(* IEC 61131-3 sources: AXOpen/src/showcase/app/src/IO, 9 files *)

(* ---- HwIdentifierList.st ---- *)
NAMESPACE AXOpen.Showcase
    TYPE HwIdentifierList : ARRAY[0..442] OF UINT :=
            [
                UINT#32,
                UINT#48,
                UINT#51,
                UINT#54,
                UINT#64,
                UINT#65,
                UINT#66,
                UINT#72,
                UINT#73,
                UINT#74,
                UINT#117,
                UINT#120,
                UINT#121,
                UINT#135,
                UINT#256,
                UINT#257,
                UINT#258,
                UINT#259,
                UINT#260,
                UINT#261,
                UINT#262,
                UINT#263,
                UINT#264,
                UINT#265,
                UINT#266,
                UINT#267,
                UINT#268,
                UINT#269,
                UINT#270,
                UINT#271,
                UINT#272,
                UINT#273,
                UINT#274,
                UINT#275,
                UINT#276,
                UINT#277,
                UINT#278,
                UINT#279,
                UINT#280,
                UINT#281,
                UINT#282,
                UINT#283,
                UINT#284,
                UINT#285,
                UINT#286,
                UINT#287,
                UINT#288,
                UINT#289,
                UINT#290,
                UINT#291,
                UINT#292,
                UINT#293,
                UINT#294,
                UINT#295,
                UINT#296,
                UINT#297,
                UINT#298,
                UINT#299,
                UINT#300,
                UINT#301,
                UINT#302,
                UINT#303,
                UINT#304,
                UINT#305,
                UINT#306,
                UINT#307,
                UINT#308,
                UINT#309,
                UINT#310,
                UINT#311,
                UINT#312,
                UINT#313,
                UINT#314,
                UINT#315,
                UINT#316,
                UINT#317,
                UINT#318,
                UINT#319,
                UINT#320,
                UINT#321,
                UINT#322,
                UINT#323,
                UINT#324,
                UINT#325,
                UINT#326,
                UINT#327,
                UINT#328,
                UINT#329,
                UINT#330,
                UINT#331,
                UINT#332,
                UINT#333,
                UINT#334,
                UINT#335,
                UINT#336,
                UINT#337,
                UINT#338,
                UINT#339,
                UINT#340,
                UINT#341,
                UINT#342,
                UINT#343,
                UINT#344,
                UINT#345,
                UINT#346,
                UINT#347,
                UINT#348,
                UINT#349,
                UINT#350,
                UINT#351,
                UINT#352,
                UINT#353,
                UINT#354,
                UINT#355,
                UINT#356,
                UINT#357,
                UINT#358,
                UINT#359,
                UINT#360,
                UINT#361,
                UINT#362,
                UINT#363,
                UINT#364,
                UINT#365,
                UINT#366,
                UINT#367,
                UINT#368,
                UINT#369,
                UINT#370,
                UINT#371,
                UINT#372,
                UINT#373,
                UINT#374,
                UINT#375,
                UINT#376,
                UINT#377,
                UINT#378,
                UINT#379,
                UINT#380,
                UINT#381,
                UINT#382,
                UINT#383,
                UINT#384,
                UINT#385,
                UINT#386,
                UINT#387,
                UINT#388,
                UINT#389,
                UINT#390,
                UINT#391,
                UINT#392,
                UINT#393,
                UINT#394,
                UINT#395,
                UINT#396,
                UINT#397,
                UINT#398,
                UINT#399,
                UINT#400,
                UINT#401,
                UINT#402,
                UINT#403,
                UINT#404,
                UINT#405,
                UINT#406,
                UINT#407,
                UINT#408,
                UINT#409,
                UINT#410,
                UINT#411,
                UINT#412,
                UINT#413,
                UINT#414,
                UINT#415,
                UINT#416,
                UINT#417,
                UINT#418,
                UINT#419,
                UINT#420,
                UINT#421,
                UINT#422,
                UINT#423,
                UINT#424,
                UINT#425,
                UINT#426,
                UINT#427,
                UINT#428,
                UINT#429,
                UINT#430,
                UINT#431,
                UINT#432,
                UINT#433,
                UINT#434,
                UINT#435,
                UINT#436,
                UINT#437,
                UINT#438,
                UINT#439,
                UINT#440,
                UINT#441,
                UINT#442,
                UINT#443,
                UINT#444,
                UINT#445,
                UINT#446,
                UINT#447,
                UINT#448,
                UINT#449,
                UINT#450,
                UINT#451,
                UINT#452,
                UINT#453,
                UINT#454,
                UINT#455,
                UINT#456,
                UINT#457,
                UINT#458,
                UINT#459,
                UINT#460,
                UINT#461,
                UINT#462,
                UINT#463,
                UINT#464,
                UINT#465,
                UINT#466,
                UINT#467,
                UINT#468,
                UINT#469,
                UINT#470,
                UINT#471,
                UINT#472,
                UINT#473,
                UINT#474,
                UINT#475,
                UINT#476,
                UINT#477,
                UINT#478,
                UINT#479,
                UINT#480,
                UINT#481,
                UINT#482,
                UINT#483,
                UINT#484,
                UINT#485,
                UINT#486,
                UINT#487,
                UINT#488,
                UINT#489,
                UINT#490,
                UINT#491,
                UINT#492,
                UINT#493,
                UINT#494,
                UINT#495,
                UINT#496,
                UINT#497,
                UINT#498,
                UINT#499,
                UINT#500,
                UINT#501,
                UINT#502,
                UINT#503,
                UINT#504,
                UINT#505,
                UINT#506,
                UINT#507,
                UINT#508,
                UINT#509,
                UINT#510,
                UINT#511,
                UINT#512,
                UINT#513,
                UINT#514,
                UINT#515,
                UINT#516,
                UINT#517,
                UINT#518,
                UINT#519,
                UINT#520,
                UINT#521,
                UINT#522,
                UINT#523,
                UINT#524,
                UINT#525,
                UINT#526,
                UINT#527,
                UINT#528,
                UINT#529,
                UINT#530,
                UINT#531,
                UINT#532,
                UINT#533,
                UINT#534,
                UINT#535,
                UINT#536,
                UINT#537,
                UINT#538,
                UINT#539,
                UINT#540,
                UINT#541,
                UINT#542,
                UINT#543,
                UINT#544,
                UINT#545,
                UINT#546,
                UINT#547,
                UINT#548,
                UINT#549,
                UINT#550,
                UINT#551,
                UINT#552,
                UINT#553,
                UINT#554,
                UINT#555,
                UINT#556,
                UINT#557,
                UINT#558,
                UINT#559,
                UINT#560,
                UINT#561,
                UINT#562,
                UINT#563,
                UINT#564,
                UINT#565,
                UINT#566,
                UINT#567,
                UINT#568,
                UINT#569,
                UINT#570,
                UINT#571,
                UINT#572,
                UINT#573,
                UINT#574,
                UINT#575,
                UINT#576,
                UINT#577,
                UINT#578,
                UINT#579,
                UINT#580,
                UINT#581,
                UINT#582,
                UINT#583,
                UINT#584,
                UINT#585,
                UINT#586,
                UINT#587,
                UINT#588,
                UINT#589,
                UINT#590,
                UINT#591,
                UINT#592,
                UINT#593,
                UINT#594,
                UINT#595,
                UINT#596,
                UINT#597,
                UINT#598,
                UINT#599,
                UINT#600,
                UINT#601,
                UINT#602,
                UINT#603,
                UINT#604,
                UINT#605,
                UINT#606,
                UINT#607,
                UINT#608,
                UINT#609,
                UINT#610,
                UINT#611,
                UINT#612,
                UINT#613,
                UINT#614,
                UINT#615,
                UINT#616,
                UINT#617,
                UINT#618,
                UINT#619,
                UINT#620,
                UINT#621,
                UINT#622,
                UINT#623,
                UINT#624,
                UINT#625,
                UINT#626,
                UINT#627,
                UINT#628,
                UINT#629,
                UINT#630,
                UINT#631,
                UINT#632,
                UINT#633,
                UINT#634,
                UINT#635,
                UINT#636,
                UINT#637,
                UINT#638,
                UINT#639,
                UINT#640,
                UINT#641,
                UINT#642,
                UINT#643,
                UINT#644,
                UINT#645,
                UINT#646,
                UINT#647,
                UINT#648,
                UINT#649,
                UINT#650,
                UINT#651,
                UINT#652,
                UINT#653,
                UINT#654,
                UINT#655,
                UINT#656,
                UINT#657,
                UINT#658,
                UINT#659,
                UINT#660,
                UINT#661,
                UINT#662,
                UINT#663,
                UINT#664,
                UINT#665,
                UINT#666,
                UINT#667,
                UINT#668,
                UINT#669,
                UINT#670,
                UINT#671,
                UINT#672,
                UINT#673,
                UINT#674,
                UINT#675,
                UINT#676,
                UINT#677,
                UINT#678,
                UINT#679,
                UINT#680,
                UINT#681,
                UINT#682,
                UINT#683,
                UINT#684
    ];
END_TYPE
END_NAMESPACE

(* ---- HwIdentifiers.st ---- *)
NAMESPACE AXOpen.Showcase
    TYPE
        HwIdentifiers : UINT
        (
            plc_line_HwID := UINT#32,
            plc_line_plc_line_HwID := UINT#48,
            plc_line_plc_line_Card_reader_writer_1_HwID := UINT#51,
            plc_line_plc_line_CPU_display_1_HwID := UINT#54,
            plc_line_plc_line_PROFINET_interface_1_HwID := UINT#64,
            plc_line_plc_line_PROFINET_interface_1_Port_1_HwID := UINT#65,
            plc_line_plc_line_PROFINET_interface_1_Port_2_HwID := UINT#66,
            plc_line_plc_line_PROFINET_interface_2_HwID := UINT#72,
            plc_line_plc_line_PROFINET_interface_2_Port_3_HwID := UINT#73,
            plc_line_plc_line_PROFINET_interface_2_Port_4_HwID := UINT#74,
            plc_line_plc_line_OPC_UA_1_HwID := UINT#117,
            plc_line_plc_line_PROFINET_interface_GBIT_3_HwID := UINT#120,
            plc_line_plc_line_PROFINET_interface_GBIT_3_Port_5_HwID := UINT#121,
            plc_line_plc_line_Virtual_communication_interface_HwID := UINT#135,
            profinet_plc_line_HwID := UINT#256,
            smc_ex260_spn_32_smc_ex260_spn_32_Interface_HwID := UINT#257,
            smc_ex260_spn_32_HwID := UINT#258,
            smc_ex260_spn_32_smc_ex260_spn_32_Interface_Port_1_HwID := UINT#259,
            smc_ex260_spn_32_smc_ex260_spn_32_Interface_Port_2_HwID := UINT#260,
            smc_ex260_spn_32_Rack_HwID := UINT#261,
            smc_ex260_spn_32_smc_ex260_spn_32_HwID := UINT#262,
            smc_ex260_spn_32_smc_ex260_spn_32_Outputs32_4_byte__Output_HwID := UINT#263,
            smc_ex260_spn_32_smc_ex260_spn_32_EX260_SPN_1_2_HwID := UINT#264,
            smc_ex260_spn_16_smc_ex260_spn_16_Interface_HwID := UINT#265,
            smc_ex260_spn_16_HwID := UINT#266,
            smc_ex260_spn_16_smc_ex260_spn_16_Interface_Port_1_HwID := UINT#267,
            smc_ex260_spn_16_smc_ex260_spn_16_Interface_Port_2_HwID := UINT#268,
            smc_ex260_spn_16_Rack_HwID := UINT#269,
            smc_ex260_spn_16_smc_ex260_spn_16_HwID := UINT#270,
            smc_ex260_spn_16_smc_ex260_spn_16_Outputs16_2_byte__Output_HwID := UINT#271,
            smc_ex260_spn_16_smc_ex260_spn_16_EX260_SPN_3_4_HwID := UINT#272,
            aes_pnio_aes_pnio_PN_IO_HwID := UINT#273,
            aes_pnio_HwID := UINT#274,
            aes_pnio_aes_pnio_PN_IO_Port_1_HwID := UINT#275,
            aes_pnio_aes_pnio_PN_IO_Port_2_HwID := UINT#276,
            aes_pnio_Rack_HwID := UINT#277,
            aes_pnio_aes_pnio_HwID := UINT#278,
            aes_pnio_Slot_1_Valve_driver_4_valves_4_HwID := UINT#279,
            aes_pnio_aes_pnio_AES_Modul_HwID := UINT#280,
            rf186c_cyc_rf186c_cyc_profinet_HwID := UINT#281,
            rf186c_cyc_HwID := UINT#282,
            rf186c_cyc_rf186c_cyc_profinet_Port_1_HwID := UINT#283,
            rf186c_cyc_rf186c_cyc_profinet_Port_2_HwID := UINT#284,
            rf186c_cyc_Rack_HwID := UINT#285,
            rf186c_cyc_rf186c_cyc_HwID := UINT#286,
            rf186c_cyc_RF340R_1_Reader_128_byte__cyclic_io_communication_HwID := UINT#287,
            rf186c_cyc_RF260R_1_Reader_32_byte__cyclic_io_communication_HwID := UINT#288,
            rf186c_cyc_rf186c_cyc_CM_Communication_HwID := UINT#289,
            rf186c_cyc_rf186c_cyc_RF186C_cyc_V2_2_HwID := UINT#290,
            et200sp_CM_4xIO_Link_RF200_et200sp_CM_4xIO_Link_RF200_profinet_HwID := UINT#291,
            et200sp_CM_4xIO_Link_RF200_HwID := UINT#292,
            et200sp_CM_4xIO_Link_RF200_et200sp_CM_4xIO_Link_RF200_Port_1_HwID := UINT#293,
            et200sp_CM_4xIO_Link_RF200_et200sp_CM_4xIO_Link_RF200_Port_2_HwID := UINT#294,
            et200sp_CM_4xIO_Link_RF200_Rack_HwID := UINT#295,
            et200sp_CM_4xIO_Link_RF200_et200sp_CM_4xIO_Link_RF200_HwID := UINT#296,
            et200sp_CM_4xIO_Link_RF200_Server_module_V1_1_Server_module_V1_1_0_bytes_HwID := UINT#297,
            et200sp_CM_4xIO_Link_RF200_CM_4xIO_Link_V2_2_144I_128O_1_CM_4xIO_Link_V2_2_144I_128O_HwID := UINT#298,
            et200sp_CM_4xIO_Link_RF200_et200sp_CM_4xIO_Link_RF200_IM_155_6_PN_ST_V4_2_HwID := UINT#299,
            rf186c_rf186c_profinet_HwID := UINT#300,
            rf186c_HwID := UINT#301,
            rf186c_rf186c_profinet_Port_1_HwID := UINT#302,
            rf186c_rf186c_profinet_Port_2_HwID := UINT#303,
            rf186c_Rack_HwID := UINT#304,
            rf186c_rf186c_HwID := UINT#305,
            rf186c_Reader_1__Reader__HwID := UINT#306,
            rf186c_rf186c_CM_1__Communication__HwID := UINT#307,
            rf186c_rf186c_RF186C_V2_x_HwID := UINT#308,
            et200sp_et200sp_profinet_HwID := UINT#309,
            et200sp_HwID := UINT#310,
            et200sp_et200sp_Port_1_HwID := UINT#311,
            et200sp_et200sp_Port_2_HwID := UINT#312,
            et200sp_Rack_HwID := UINT#313,
            et200sp_et200sp_HwID := UINT#314,
            et200sp_Server_module_V1_1_Server_module_V1_1_0_bytes_HwID := UINT#315,
            et200sp_CpPtp_CM_PtP_V2_0_HwID := UINT#316,
            et200sp_et200sp_IM_155_6_PN_ST_V4_2_HwID := UINT#317,
            BNIPNT507005Z040_BNIPNT507005Z040_profinet_HwID := UINT#318,
            BNIPNT507005Z040_HwID := UINT#319,
            BNIPNT507005Z040_BNIPNT507005Z040_profinet_port_1_M12_HwID := UINT#320,
            BNIPNT507005Z040_BNIPNT507005Z040_profinet_port_2_M12_HwID := UINT#321,
            BNIPNT507005Z040_Rack_HwID := UINT#322,
            BNIPNT507005Z040_BNIPNT507005Z040_HwID := UINT#323,
            BNIPNT507005Z040_BIS_M_4XX_045_1_BIS_M_4XX_045_HwID := UINT#324,
            BNIPNT507005Z040_Standard_I_O_4_Standard_I_O_HwID := UINT#325,
            BNIPNT507005Z040_Standard_I_O_3_Standard_I_O_HwID := UINT#326,
            BNIPNT507005Z040_Standard_I_O_2_Standard_I_O_HwID := UINT#327,
            BNIPNT507005Z040_BNIPNT507005Z040_BNI_PNT_507_005_Z040_HwID := UINT#328,
            rexroth_cs351_rexroth_cs351_Interface_HwID := UINT#329,
            rexroth_cs351_HwID := UINT#330,
            rexroth_cs351_rexroth_cs351_Interface_Port_1_HwID := UINT#331,
            rexroth_cs351_Rack_HwID := UINT#332,
            rexroth_cs351_rexroth_cs351_HwID := UINT#333,
            rexroth_cs351_Input_2_word_1_Input_2_word_HwID := UINT#334,
            rexroth_cs351_Input_4_word_16_Input_4_word_HwID := UINT#335,
            rexroth_cs351_Input_4_word_15_Input_4_word_HwID := UINT#336,
            rexroth_cs351_Input_4_word_14_Input_4_word_HwID := UINT#337,
            rexroth_cs351_Input_4_word_13_Input_4_word_HwID := UINT#338,
            rexroth_cs351_Input_4_word_12_Input_4_word_HwID := UINT#339,
            rexroth_cs351_Input_4_word_11_Input_4_word_HwID := UINT#340,
            rexroth_cs351_Input_4_word_10_Input_4_word_HwID := UINT#341,
            rexroth_cs351_Input_4_word_9_Input_4_word_HwID := UINT#342,
            rexroth_cs351_Input_4_word_8_Input_4_word_HwID := UINT#343,
            rexroth_cs351_Input_4_word_7_Input_4_word_HwID := UINT#344,
            rexroth_cs351_Input_4_word_6_Input_4_word_HwID := UINT#345,
            rexroth_cs351_Input_4_word_5_Input_4_word_HwID := UINT#346,
            rexroth_cs351_Input_4_word_4_Input_4_word_HwID := UINT#347,
            rexroth_cs351_Input_4_word_3_Input_4_word_HwID := UINT#348,
            rexroth_cs351_Input_4_word_2_Input_4_word_HwID := UINT#349,
            rexroth_cs351_Input_4_word_1_Input_4_word_HwID := UINT#350,
            rexroth_cs351_Output_2_word_1_Output_2_word_HwID := UINT#351,
            rexroth_cs351_Output_4_word_8_Output_4_word_HwID := UINT#352,
            rexroth_cs351_Output_4_word_7_Output_4_word_HwID := UINT#353,
            rexroth_cs351_Output_4_word_6_Output_4_word_HwID := UINT#354,
            rexroth_cs351_Output_4_word_5_Output_4_word_HwID := UINT#355,
            rexroth_cs351_Output_4_word_4_Output_4_word_HwID := UINT#356,
            rexroth_cs351_Output_4_word_3_Output_4_word_HwID := UINT#357,
            rexroth_cs351_Output_4_word_2_Output_4_word_HwID := UINT#358,
            rexroth_cs351_Output_4_word_1_Output_4_word_HwID := UINT#359,
            rexroth_cs351_rexroth_cs351_DAP_V2_0_HwID := UINT#360,
            rexroth_press_rexroth_press_PN_IO_HwID := UINT#361,
            rexroth_press_HwID := UINT#362,
            rexroth_press_rexroth_press_PN_IO_Port_1_HwID := UINT#363,
            rexroth_press_rexroth_press_PN_IO_Port_2_HwID := UINT#364,
            rexroth_press_Rack_HwID := UINT#365,
            rexroth_press_rexroth_press_HwID := UINT#366,
            rexroth_press_Output_21_Words_ID_OutMod_21Words_HwID := UINT#367,
            rexroth_press_Input_24_Words_ID_InMod_24Words_HwID := UINT#368,
            rexroth_press_ParamCh_5Words_ID_PaCh_5Words_HwID := UINT#369,
            rexroth_press_F_Modul_not_used_ID_FMod_NotUsed_HwID := UINT#370,
            rexroth_press_rexroth_press_DAP_1_HwID := UINT#371,
            dukaneiqauto_dukaneiqauto_Interface_HwID := UINT#372,
            dukaneiqauto_HwID := UINT#373,
            dukaneiqauto_dukaneiqauto_Interface_Port_1_HwID := UINT#374,
            dukaneiqauto_dukaneiqauto_Interface_Port_2_HwID := UINT#375,
            dukaneiqauto_Rack_HwID := UINT#376,
            dukaneiqauto_dukaneiqauto_HwID := UINT#377,
            dukaneiqauto_PLC_to_iQ_Outputs_PLC_to_iQ_Outputs_HwID := UINT#378,
            dukaneiqauto_iQ_to_PLC_Inputs_iQ_to_PLC_Inputs_HwID := UINT#379,
            dukaneiqauto_dukaneiqauto_DAP_HwID := UINT#380,
            desoutter_cvic_ii_desoutter_cvic_ii_Interface_HwID := UINT#381,
            desoutter_cvic_ii_HwID := UINT#382,
            desoutter_cvic_ii_desoutter_cvic_ii_Interface_Port_1_HwID := UINT#383,
            desoutter_cvic_ii_Rack_HwID := UINT#384,
            desoutter_cvic_ii_desoutter_cvic_ii_HwID := UINT#385,
            desoutter_cvic_ii_Output_1_byte_2_Output_1_byte_HwID := UINT#386,
            desoutter_cvic_ii_Output_1_byte_1_Output_1_byte_HwID := UINT#387,
            desoutter_cvic_ii_Input_1_word_2_Input_1_word_HwID := UINT#388,
            desoutter_cvic_ii_Input_2_word_2_Input_2_word_HwID := UINT#389,
            desoutter_cvic_ii_Input_1_word_1_Input_1_word_HwID := UINT#390,
            desoutter_cvic_ii_Input_2_word_1_Input_2_word_HwID := UINT#391,
            desoutter_cvic_ii_Input_1_byte_2_Input_1_byte_HwID := UINT#392,
            desoutter_cvic_ii_Input_1_byte_1_Input_1_byte_HwID := UINT#393,
            desoutter_cvic_ii_desoutter_cvic_ii_RT_HwID := UINT#394,
            zebra_zebra_Interface_HwID := UINT#395,
            zebra_HwID := UINT#396,
            zebra_zebra_Interface_Port_1_HwID := UINT#397,
            zebra_Rack_HwID := UINT#398,
            zebra_zebra_HwID := UINT#399,
            zebra_Data88Bin6Bout_Data_and_Transfer_Control_v2_HwID := UINT#400,
            zebra_zebra_EA3600_PIO_Interface_HwID := UINT#401,
            keyence_iv3_keyence_iv3_Interface_HwID := UINT#402,
            keyence_iv3_HwID := UINT#403,
            keyence_iv3_keyence_iv3_Interface_Port_1_HwID := UINT#404,
            keyence_iv3_Rack_HwID := UINT#405,
            keyence_iv3_keyence_iv3_HwID := UINT#406,
            keyence_iv3_DeviceResultBits_2_Device_Result_Bits_HwID := UINT#407,
            keyence_iv3_ToolResult_64_Tool_Result_HwID := UINT#408,
            keyence_iv3_ToolResult_63_Tool_Result_HwID := UINT#409,
            keyence_iv3_ToolResult_62_Tool_Result_HwID := UINT#410,
            keyence_iv3_ToolResult_61_Tool_Result_HwID := UINT#411,
            keyence_iv3_ToolResult_60_Tool_Result_HwID := UINT#412,
            keyence_iv3_ToolResult_59_Tool_Result_HwID := UINT#413,
            keyence_iv3_ToolResult_58_Tool_Result_HwID := UINT#414,
            keyence_iv3_ToolResult_57_Tool_Result_HwID := UINT#415,
            keyence_iv3_ToolResult_56_Tool_Result_HwID := UINT#416,
            keyence_iv3_ToolResult_55_Tool_Result_HwID := UINT#417,
            keyence_iv3_ToolResult_54_Tool_Result_HwID := UINT#418,
            keyence_iv3_ToolResult_53_Tool_Result_HwID := UINT#419,
            keyence_iv3_ToolResult_52_Tool_Result_HwID := UINT#420,
            keyence_iv3_ToolResult_51_Tool_Result_HwID := UINT#421,
            keyence_iv3_ToolResult_50_Tool_Result_HwID := UINT#422,
            keyence_iv3_ToolResult_49_Tool_Result_HwID := UINT#423,
            keyence_iv3_ToolResult_48_Tool_Result_HwID := UINT#424,
            keyence_iv3_ToolResult_47_Tool_Result_HwID := UINT#425,
            keyence_iv3_ToolResult_46_Tool_Result_HwID := UINT#426,
            keyence_iv3_ToolResult_45_Tool_Result_HwID := UINT#427,
            keyence_iv3_ToolResult_44_Tool_Result_HwID := UINT#428,
            keyence_iv3_ToolResult_43_Tool_Result_HwID := UINT#429,
            keyence_iv3_ToolResult_42_Tool_Result_HwID := UINT#430,
            keyence_iv3_ToolResult_41_Tool_Result_HwID := UINT#431,
            keyence_iv3_ToolResult_40_Tool_Result_HwID := UINT#432,
            keyence_iv3_ToolResult_39_Tool_Result_HwID := UINT#433,
            keyence_iv3_ToolResult_38_Tool_Result_HwID := UINT#434,
            keyence_iv3_ToolResult_37_Tool_Result_HwID := UINT#435,
            keyence_iv3_ToolResult_36_Tool_Result_HwID := UINT#436,
            keyence_iv3_ToolResult_35_Tool_Result_HwID := UINT#437,
            keyence_iv3_ToolResult_34_Tool_Result_HwID := UINT#438,
            keyence_iv3_ToolResult_33_Tool_Result_HwID := UINT#439,
            keyence_iv3_ToolResult_32_Tool_Result_HwID := UINT#440,
            keyence_iv3_ToolResult_31_Tool_Result_HwID := UINT#441,
            keyence_iv3_ToolResult_30_Tool_Result_HwID := UINT#442,
            keyence_iv3_ToolResult_29_Tool_Result_HwID := UINT#443,
            keyence_iv3_ToolResult_28_Tool_Result_HwID := UINT#444,
            keyence_iv3_ToolResult_27_Tool_Result_HwID := UINT#445,
            keyence_iv3_ToolResult_26_Tool_Result_HwID := UINT#446,
            keyence_iv3_ToolResult_25_Tool_Result_HwID := UINT#447,
            keyence_iv3_ToolResult_24_Tool_Result_HwID := UINT#448,
            keyence_iv3_ToolResult_23_Tool_Result_HwID := UINT#449,
            keyence_iv3_ToolResult_22_Tool_Result_HwID := UINT#450,
            keyence_iv3_ToolResult_21_Tool_Result_HwID := UINT#451,
            keyence_iv3_ToolResult_20_Tool_Result_HwID := UINT#452,
            keyence_iv3_ToolResult_19_Tool_Result_HwID := UINT#453,
            keyence_iv3_ToolResult_18_Tool_Result_HwID := UINT#454,
            keyence_iv3_ToolResult_17_Tool_Result_HwID := UINT#455,
            keyence_iv3_ToolResult_16_Tool_Result_HwID := UINT#456,
            keyence_iv3_ToolResult_15_Tool_Result_HwID := UINT#457,
            keyence_iv3_ToolResult_14_Tool_Result_HwID := UINT#458,
            keyence_iv3_ToolResult_13_Tool_Result_HwID := UINT#459,
            keyence_iv3_ToolResult_12_Tool_Result_HwID := UINT#460,
            keyence_iv3_ToolResult_11_Tool_Result_HwID := UINT#461,
            keyence_iv3_ToolResult_10_Tool_Result_HwID := UINT#462,
            keyence_iv3_ToolResult_9_Tool_Result_HwID := UINT#463,
            keyence_iv3_ToolResult_8_Tool_Result_HwID := UINT#464,
            keyence_iv3_ToolResult_7_Tool_Result_HwID := UINT#465,
            keyence_iv3_ToolResult_6_Tool_Result_HwID := UINT#466,
            keyence_iv3_ToolResult_5_Tool_Result_HwID := UINT#467,
            keyence_iv3_ToolResult_4_Tool_Result_HwID := UINT#468,
            keyence_iv3_ToolResult_3_Tool_Result_HwID := UINT#469,
            keyence_iv3_ToolResult_2_Tool_Result_HwID := UINT#470,
            keyence_iv3_ToolResult_1_Tool_Result_HwID := UINT#471,
            keyence_iv3_PositionAdjustResult_Position_Adjust_Result_HwID := UINT#472,
            keyence_iv3_DeviceStatistics_Device_Statistics_HwID := UINT#473,
            keyence_iv3_DeviceStatusWords_Device_Status_Words_HwID := UINT#474,
            keyence_iv3_DeviceResultBits_1_Device_Result_Bits_HwID := UINT#475,
            keyence_iv3_CommandStatusBits_Command_Status_Bits_HwID := UINT#476,
            keyence_iv3_CommandControl_Command_Control_HwID := UINT#477,
            keyence_iv3_keyence_iv3_IV3_XXXX_HwID := UINT#478,
            keyence_sr_1000_keyence_sr_1000_Interface_HwID := UINT#479,
            keyence_sr_1000_HwID := UINT#480,
            keyence_sr_1000_keyence_sr_1000_Interface_Port_1_HwID := UINT#481,
            keyence_sr_1000_Rack_HwID := UINT#482,
            keyence_sr_1000_keyence_sr_1000_HwID := UINT#483,
            keyence_sr_1000_UserData_128_User_Data_128Byte_HwID := UINT#484,
            keyence_sr_1000_ParameterBank_Parameter_Bank_Number_HwID := UINT#485,
            keyence_sr_1000_CompletionClearControl_Completion_Clear_Control_Bits_HwID := UINT#486,
            keyence_sr_1000_OperationInstructionControl_Operation_instruction_Control_Bits_HwID := UINT#487,
            keyence_sr_1000_LatchAndErrorClearControl_Latch_and_Error_Clear_Control_Bits_HwID := UINT#488,
            keyence_sr_1000_ResultData_128_Read_Data_128Byte_HwID := UINT#489,
            keyence_sr_1000_OperationResultStatus_Operation_Result_Status_HwID := UINT#490,
            keyence_sr_1000_MatchingLevelAndTotalEvaluationGradeStatus_Matching_Level_and_Total_Evaluation_Grade_Status_HwID := UINT#491,
            keyence_sr_1000_UnstableReadStatus_Unstable_Read_Status_Bits_HwID := UINT#492,
            keyence_sr_1000_TerminalStatus_Terminal_Status_Bits_HwID := UINT#493,
            keyence_sr_1000_ErrorStatus_Error_Status_Bits_HwID := UINT#494,
            keyence_sr_1000_CompletionStatus_Completion_Status_Bits_HwID := UINT#495,
            keyence_sr_1000_BusyStatus_BUSY_Status_Bits_HwID := UINT#496,
            keyence_sr_1000_HandshakeAndGeneralErrorStatus_Handshake_and_General_Error_Status_Bits_HwID := UINT#497,
            keyence_sr_1000_keyence_sr_1000_SR_1000X_HwID := UINT#498,
            keyence_sr_750_keyence_sr_750_Interface_HwID := UINT#499,
            keyence_sr_750_HwID := UINT#500,
            keyence_sr_750_keyence_sr_750_Interface_Port_1_HwID := UINT#501,
            keyence_sr_750_Rack_HwID := UINT#502,
            keyence_sr_750_keyence_sr_750_HwID := UINT#503,
            keyence_sr_750_UserData_128_User_Data_128Byte_HwID := UINT#504,
            keyence_sr_750_ParameterBank_Parameter_Bank_Number_HwID := UINT#505,
            keyence_sr_750_CompletionClearControl_Completion_Clear_Control_Bits_HwID := UINT#506,
            keyence_sr_750_OperationInstructionControl_Operation_instruction_Control_Bits_HwID := UINT#507,
            keyence_sr_750_LatchAndErrorClearControl_Latch_and_Error_Clear_Control_Bits_HwID := UINT#508,
            keyence_sr_750_ResultData_128_Read_Data_128Byte_HwID := UINT#509,
            keyence_sr_750_OperationResultStatus_Operation_Result_Status_HwID := UINT#510,
            keyence_sr_750_MatchingLevelAndTotalEvaluationGradeStatus_Matching_Level_and_Total_Evaluation_Grade_Status_HwID := UINT#511,
            keyence_sr_750_UnstableReadStatus_Unstable_Read_Status_Bits_HwID := UINT#512,
            keyence_sr_750_TerminalStatus_Terminal_Status_Bits_HwID := UINT#513,
            keyence_sr_750_ErrorStatus_Error_Status_Bits_HwID := UINT#514,
            keyence_sr_750_CompletionStatus_Completion_Status_Bits_HwID := UINT#515,
            keyence_sr_750_BusyStatus_BUSY_Status_Bits_HwID := UINT#516,
            keyence_sr_750_HandshakeAndGeneralErrorStatus_Handshake_and_General_Error_Status_Bits_HwID := UINT#517,
            keyence_sr_750_keyence_sr_750_SR_75X_HwID := UINT#518,
            vision_pro_vision_pro_Interface_HwID := UINT#519,
            vision_pro_HwID := UINT#520,
            vision_pro_vision_pro_Interface_Port_1_HwID := UINT#521,
            vision_pro_Rack_HwID := UINT#522,
            vision_pro_vision_pro_HwID := UINT#523,
            vision_pro_Result_Data_64_bytes_1_Results_64_bytes_HwID := UINT#524,
            vision_pro_Result_Data_240_bytes_5_Results_240_bytes_HwID := UINT#525,
            vision_pro_Result_Data_240_bytes_4_Results_240_bytes_HwID := UINT#526,
            vision_pro_Result_Data_240_bytes_3_Results_240_bytes_HwID := UINT#527,
            vision_pro_Result_Data_240_bytes_2_Results_240_bytes_HwID := UINT#528,
            vision_pro_User_Data_64_bytes_1_User_Data_64_bytes_HwID := UINT#529,
            vision_pro_User_Data_240_bytes_5_User_Data_240_bytes_HwID := UINT#530,
            vision_pro_User_Data_240_bytes_4_User_Data_240_bytes_HwID := UINT#531,
            vision_pro_User_Data_240_bytes_3_User_Data_240_bytes_HwID := UINT#532,
            vision_pro_User_Data_240_bytes_2_User_Data_240_bytes_HwID := UINT#533,
            vision_pro_Result_Data_240_bytes_1_Results_240_bytes_HwID := UINT#534,
            vision_pro_User_Data_240_bytes_1_User_Data_240_bytes_HwID := UINT#535,
            vision_pro_Engine_Control_4_Engine_Control_HwID := UINT#536,
            vision_pro_Engine_Control_3_Engine_Control_HwID := UINT#537,
            vision_pro_Engine_Control_2_Engine_Control_HwID := UINT#538,
            vision_pro_Engine_Control_1_Engine_Control_HwID := UINT#539,
            vision_pro_System_Control_System_Control_HwID := UINT#540,
            vision_pro_vision_pro_Communication_Card_CC24_HwID := UINT#541,
            cognex_insight_2800_cognex_insight_2800_Interface_HwID := UINT#542,
            cognex_insight_2800_HwID := UINT#543,
            cognex_insight_2800_cognex_insight_2800_Interface_Port_1_HwID := UINT#544,
            cognex_insight_2800_Rack_HwID := UINT#545,
            cognex_insight_2800_cognex_insight_2800_HwID := UINT#546,
            cognex_insight_2800_Slot_14_Results_250_bytes_HwID := UINT#547,
            cognex_insight_2800_Slot_13_Results_250_bytes_HwID := UINT#548,
            cognex_insight_2800_Slot_12_Results_250_bytes_HwID := UINT#549,
            cognex_insight_2800_Slot_11_ResultData_250_Results_250_bytes_HwID := UINT#550,
            cognex_insight_2800_Slot_9_User_Data_254_bytes_HwID := UINT#551,
            cognex_insight_2800_Slot_8_User_Data_254_bytes_HwID := UINT#552,
            cognex_insight_2800_Slot_7_User_Data_254_bytes_HwID := UINT#553,
            cognex_insight_2800_Slot_2_Acquisition_Status_HwID := UINT#554,
            cognex_insight_2800_Slot_4_Inspection_Status_HwID := UINT#555,
            cognex_insight_2800_Slot_5_Command_Control_HwID := UINT#556,
            cognex_insight_2800_Slot_6_ExternalEvent_Control_HwID := UINT#557,
            cognex_insight_2800_Slot_3_Inspection_Control_HwID := UINT#558,
            cognex_insight_2800_Slot_1_Acquisition_Control_HwID := UINT#559,
            cognex_insight_2800_cognex_insight_2800_In_Sight_IS28XX_CC_B_HwID := UINT#560,
            cognex_dataman_380_cognex_dataman_380_Interface_HwID := UINT#561,
            cognex_dataman_380_HwID := UINT#562,
            cognex_dataman_380_cognex_dataman_380_Interface_Port_1_HwID := UINT#563,
            cognex_dataman_380_Rack_HwID := UINT#564,
            cognex_dataman_380_cognex_dataman_380_HwID := UINT#565,
            cognex_dataman_380_ResultData_128_Result_Data_128_bytes_HwID := UINT#566,
            cognex_dataman_380_UserData_128_User_Data_128_bytes_HwID := UINT#567,
            cognex_dataman_380_Results_Status_Results_Status_HwID := UINT#568,
            cognex_dataman_380_Acquisition_Status_Acquisition_Status_HwID := UINT#569,
            cognex_dataman_380_Soft_Event_Control_Soft_Event_Control_HwID := UINT#570,
            cognex_dataman_380_Results_Control_Results_Control_HwID := UINT#571,
            cognex_dataman_380_Acquisition_Control_Acquisition_Control_HwID := UINT#572,
            cognex_dataman_380_cognex_dataman_380_DataMan_380_CC_B_HwID := UINT#573,
            cognex_dataman_280_cognex_dataman_280_Interface_HwID := UINT#574,
            cognex_dataman_280_HwID := UINT#575,
            cognex_dataman_280_cognex_dataman_280_Interface_Port_1_HwID := UINT#576,
            cognex_dataman_280_Rack_HwID := UINT#577,
            cognex_dataman_280_cognex_dataman_280_HwID := UINT#578,
            cognex_dataman_280_ResultData_128_Result_Data_128_bytes_HwID := UINT#579,
            cognex_dataman_280_UserData_128_User_Data_128_bytes_HwID := UINT#580,
            cognex_dataman_280_Results_Status_Results_Status_HwID := UINT#581,
            cognex_dataman_280_Acquisition_Status_Acquisition_Status_HwID := UINT#582,
            cognex_dataman_280_Soft_Event_Control_Soft_Event_Control_HwID := UINT#583,
            cognex_dataman_280_Results_Control_Results_Control_HwID := UINT#584,
            cognex_dataman_280_Acquisition_Control_Acquisition_Control_HwID := UINT#585,
            cognex_dataman_280_cognex_dataman_280_DataMan_280_CC_B_HwID := UINT#586,
            cognex_insight_7600_cognex_insight_7600_Interface_HwID := UINT#587,
            cognex_insight_7600_HwID := UINT#588,
            cognex_insight_7600_cognex_insight_7600_Interface_Port_1_HwID := UINT#589,
            cognex_insight_7600_Rack_HwID := UINT#590,
            cognex_insight_7600_cognex_insight_7600_HwID := UINT#591,
            cognex_insight_7600_ResultData_128_Results_128_bytes_HwID := UINT#592,
            cognex_insight_7600_UserData_128_User_Data_128_bytes_HwID := UINT#593,
            cognex_insight_7600_Inspection_Status_Inspection_Status_HwID := UINT#594,
            cognex_insight_7600_Acquisition_Status_Acquisition_Status_HwID := UINT#595,
            cognex_insight_7600_Command_Control_Command_Control_HwID := UINT#596,
            cognex_insight_7600_SoftEvent_Control_SoftEvent_Control_HwID := UINT#597,
            cognex_insight_7600_Inspection_Control_Inspection_Control_HwID := UINT#598,
            cognex_insight_7600_Acquisition_Control_Acquisition_Control_HwID := UINT#599,
            cognex_insight_7600_cognex_insight_7600_In_Sight_IS79XX_IS75XX_CC_B_HwID := UINT#600,
            rexroth_ctrlx_drive_rexroth_ctrlx_drive_XCS_interface_PF30_HwID := UINT#601,
            rexroth_ctrlx_drive_HwID := UINT#602,
            rexroth_ctrlx_drive_rexroth_ctrlx_drive_XCS_interface_PF30_Port_1_HwID := UINT#603,
            rexroth_ctrlx_drive_rexroth_ctrlx_drive_XCS_interface_PF30_Port_2_HwID := UINT#604,
            rexroth_ctrlx_drive_Rack_HwID := UINT#605,
            rexroth_ctrlx_drive_rexroth_ctrlx_drive_HwID := UINT#606,
            rexroth_ctrlx_drive_Outputs_HwID := UINT#607,
            rexroth_ctrlx_drive_Inputs_HwID := UINT#608,
            rexroth_ctrlx_drive_S_0_0386_0_0__Position_controller__Position_actual_value_HwID := UINT#609,
            rexroth_ctrlx_drive_S_0_0535_0_0__Velocity_controller__Velocity_actual_value_HwID := UINT#610,
            rexroth_ctrlx_drive_S_0_0390_0_0__Diagnostic_message__Manufacturer_status_register_HwID := UINT#611,
            rexroth_ctrlx_drive_S_0_0135_0_0__Drive_status_word__Value_HwID := UINT#612,
            rexroth_ctrlx_drive_S_0_0144_0_0__Signal_status_word__Value_HwID := UINT#613,
            rexroth_ctrlx_drive_S_0_1720_0_2__Power_supply_control__Status_word_HwID := UINT#614,
            rexroth_ctrlx_drive_S_0_0084_0_0__Torque_force_feedback_value_HwID := UINT#615,
            rexroth_ctrlx_drive_P_0_0106_0_0__STO_function__Operating_status_HwID := UINT#616,
            rexroth_ctrlx_drive_S_0_0134_0_0__Master_control_word__Value_HwID := UINT#617,
            rexroth_ctrlx_drive_S_0_0260_0_0__Positioning_profile__Acceleration_HwID := UINT#618,
            rexroth_ctrlx_drive_S_0_0282_0_0__Drive_controlled_positioning__Command_value_HwID := UINT#619,
            rexroth_ctrlx_drive_S_0_0359_0_0__Positioning_profile__Deceleration_HwID := UINT#620,
            rexroth_ctrlx_drive_S_0_0259_0_0__Positioning_profile__Profile_velocity_HwID := UINT#621,
            rexroth_ctrlx_drive_S_0_0145_0_0__Signal_control_word__Value_HwID := UINT#622,
            rexroth_ctrlx_drive_S_0_1720_0_1__Power_supply_control__Control_word_HwID := UINT#623,
            rexroth_ctrlx_drive_S_0_0092_0_0__Torque_force_limitation__Limit_value_bipolar_HwID := UINT#624,
            rexroth_ctrlx_drive_S_0_0080_0_0__Torque_force_command_value_HwID := UINT#625,
            rexroth_ctrlx_drive_S_0_0193_0_0__Positioning_jerk_HwID := UINT#626,
            rexroth_ctrlx_drive_rexroth_ctrlx_drive_ctrlX_DRIVE_XCS_HwID := UINT#627,
            rexroth_indradrive_rexroth_indradrive_PN_IO_HwID := UINT#628,
            rexroth_indradrive_HwID := UINT#629,
            rexroth_indradrive_rexroth_indradrive_PN_IO_Port_1_HwID := UINT#630,
            rexroth_indradrive_rexroth_indradrive_PN_IO_Port_2_HwID := UINT#631,
            rexroth_indradrive_Rack_HwID := UINT#632,
            rexroth_indradrive_rexroth_indradrive_HwID := UINT#633,
            rexroth_indradrive_Output_13_Words_ID_OutMod_13Words_HwID := UINT#634,
            rexroth_indradrive_Input_9_Words_ID_InMod_9Words_HwID := UINT#635,
            rexroth_indradrive_ParamCh_5Words_ID_PaCh_5Words_HwID := UINT#636,
            rexroth_indradrive_F_Modul_not_used_ID_FMod_NotUsed_HwID := UINT#637,
            rexroth_indradrive_rexroth_indradrive_DAP_1_HwID := UINT#638,
            festo_cmmtas_festo_cmmtas_PN_IO_Interface_HwID := UINT#639,
            festo_cmmtas_HwID := UINT#640,
            festo_cmmtas_festo_cmmtas_PN_IO_Interface_Port_1_HwID := UINT#641,
            festo_cmmtas_festo_cmmtas_PN_IO_Interface_Port_2_HwID := UINT#642,
            festo_cmmtas_Rack_HwID := UINT#643,
            festo_cmmtas_festo_cmmtas_HwID := UINT#644,
            festo_cmmtas_festo_cmmtas_DoServo_HwID := UINT#645,
            festo_cmmtas_festo_cmmtas_DoServo_Module_Access_Point_HwID := UINT#646,
            festo_cmmtas_festo_cmmtas_empty_submodule_1_HwID := UINT#647,
            festo_cmmtas_empty_submodule_HwID := UINT#648,
            festo_cmmtas_SiemensTelegram111_PZD_12_12_HwID := UINT#649,
            festo_cmmtas_SiemensTelegram750_PZD_4_1_HwID := UINT#650,
            festo_cmmtas_festo_cmmtas_CMMT_AS___MP_HwID := UINT#651,
            ureol2l_ureol2l_Interface_HwID := UINT#652,
            ureol2l_HwID := UINT#653,
            ureol2l_ureol2l_Interface_Port_1_HwID := UINT#654,
            ureol2l_Rack_HwID := UINT#655,
            ureol2l_ureol2l_HwID := UINT#656,
            ureol2l_10_O2T_General_Purpose_Registers_2_10_O2T_General_Purpose_Registers_2_HwID := UINT#657,
            ureol2l_9_O2T_General_Purpose_Registers_1_9_O2T_General_Purpose_Registers_1_HwID := UINT#658,
            ureol2l_8_O2T_Robot_IO_8_O2T_Robot_IO_HwID := UINT#659,
            ureol2l_7_T2O_General_Purpose_Float_Registers_7_T2O_General_Purpose_Float_Registers_HwID := UINT#660,
            ureol2l_6_T2O_General_Purpose_Int_Registers_6_T2O_General_Purpose_Int_Registers_HwID := UINT#661,
            ureol2l_5_T2O_General_Purpose_Bit_Registers_5_T2O_General_Purpose_Bit_Registers_HwID := UINT#662,
            ureol2l_4_T2O_TCP_4_T2O_TCP_HwID := UINT#663,
            ureol2l_3_T2O_Joints_3_T2O_Joints_HwID := UINT#664,
            ureol2l_2_T2O_IO_2_T2O_IO_HwID := UINT#665,
            ureol2l_1_T2O_State_1_T2O_State_HwID := UINT#666,
            ureol2l_ureol2l_V1_0_HwID := UINT#667,
            mitsubishi_tz535_robot_mitsubishi_tz535_robot_Interface_HwID := UINT#668,
            mitsubishi_tz535_robot_HwID := UINT#669,
            mitsubishi_tz535_robot_mitsubishi_tz535_robot_Interface_Port_1_HwID := UINT#670,
            mitsubishi_tz535_robot_mitsubishi_tz535_robot_Interface_Port_2_HwID := UINT#671,
            mitsubishi_tz535_robot_Rack_HwID := UINT#672,
            mitsubishi_tz535_robot_mitsubishi_tz535_robot_HwID := UINT#673,
            mitsubishi_tz535_robot_In_Out_64_byte_In_Out__64_byte_HwID := UINT#674,
            mitsubishi_tz535_robot_mitsubishi_tz535_robot_2D_TZ535_PNPROFINET_IO_HwID := UINT#675,
            kuka_rb2_kuka_rb2_Interface1_HwID := UINT#676,
            kuka_rb2_HwID := UINT#677,
            kuka_rb2_kuka_rb2_Interface1_Port_1_HwID := UINT#678,
            kuka_rb2_kuka_rb2_Interface1_Port_2_HwID := UINT#679,
            kuka_rb2_kuka_rb2_Interface1_Port_3_HwID := UINT#680,
            kuka_rb2_kuka_rb2_Interface1_Port_4_HwID := UINT#681,
            kuka_rb2_Rack_HwID := UINT#682,
            kuka_rb2_kuka_rb2_HwID := UINT#683,
            kuka_rb2_DIO512_512_digital_in__and_outputs_HwID := UINT#684,
            kuka_rb2_kuka_rb2_KUKA_PROFINET_6_0_HwID := UINT#685,
            kuka_rb1_kuka_rb1_Interface1_HwID := UINT#686,
            kuka_rb1_HwID := UINT#687,
            kuka_rb1_kuka_rb1_Interface1_Port_1_HwID := UINT#688,
            kuka_rb1_Rack_HwID := UINT#689,
            kuka_rb1_kuka_rb1_HwID := UINT#690,
            kuka_rb1_DIO512_512_digital_in__and_outputs_HwID := UINT#691,
            kuka_rb1_kuka_rb1_KRC4_ProfiNet_5_0_HwID := UINT#692,
            abb_omnicore_robot_abb_omnicore_robot_PROFINET_Interface_HwID := UINT#693,
            abb_omnicore_robot_HwID := UINT#694,
            abb_omnicore_robot_abb_omnicore_robot_PROFINET_Interface_Port_1_HwID := UINT#695,
            abb_omnicore_robot_Rack_HwID := UINT#696,
            abb_omnicore_robot_abb_omnicore_robot_HwID := UINT#697,
            abb_omnicore_robot_DO_64_bytes_DO_64_bytes_HwID := UINT#698,
            abb_omnicore_robot_DI_64_bytes_DI_64_bytes_HwID := UINT#699,
            abb_omnicore_robot_abb_omnicore_robot_OmniCore_Standard_PROFINET_Device_HwID := UINT#700,
            abb_irc5_robot_abb_irc5_robot_PROFINET_Interface_HwID := UINT#701,
            abb_irc5_robot_HwID := UINT#702,
            abb_irc5_robot_abb_irc5_robot_PROFINET_Interface_Port_1_HwID := UINT#703,
            abb_irc5_robot_Rack_HwID := UINT#704,
            abb_irc5_robot_abb_irc5_robot_HwID := UINT#705,
            abb_irc5_robot_DO_64_bytes_DO_64_bytes_HwID := UINT#706,
            abb_irc5_robot_DI_64_bytes_DI_64_bytes_HwID := UINT#707,
            abb_irc5_robot_abb_irc5_robot_Robot_Basic_Device_HwID := UINT#708,
            plc_line_Rail_0_HwID := UINT#709,
            plc_line_A1_A1_HwID := UINT#710
        );
    END_TYPE
END_NAMESPACE

(* ---- Inputs.st ---- *)
NAMESPACE AXOpen.Showcase
    TYPE
        {S7.extern=ReadWrite}
        {#ix-attr:[Container(Layout.Wrap)]}
        Inputs : STRUCT
	        // Module abb_irc5_robot/DI_64_bytes
	        abb_irc5_robot_DI_64_bytes_Input AT %B6025 : abb_irc5_robot_DI_64_bytes_Input_Layout;

	        // Module abb_omnicore_robot/DI_64_bytes
	        abb_omnicore_robot_DI_64_bytes_Input AT %B5961 : abb_omnicore_robot_DI_64_bytes_Input_Layout;

	        // Module BNIPNT507005Z040/BIS_M-4XX-045_1
	        BNIPNT507005Z040_BIS_M_4XX_045_1_Input AT %B318 : BNIPNT507005Z040_BIS_M_4XX_045_1_Input_Layout;

	        // Module cognex_dataman_280/Acquisition_Status
	        cognex_dataman_280_Acquisition_Status_Input AT %B5067 : cognex_dataman_280_Acquisition_Status_Input_Layout;

	        // Module cognex_dataman_280/ResultData_128
	        cognex_dataman_280_ResultData_128_Input AT %B4930 : cognex_dataman_280_ResultData_128_Input_Layout;

	        // Module cognex_dataman_280/Results_Status
	        cognex_dataman_280_Results_Status_Input AT %B5066 : cognex_dataman_280_Results_Status_Input_Layout;

	        // Module cognex_dataman_280/Soft_Event_Control
	        cognex_dataman_280_Soft_Event_Control_Input AT %B5070 : cognex_dataman_280_Soft_Event_Control_Input_Layout;

	        // Module cognex_dataman_380/Acquisition_Status
	        cognex_dataman_380_Acquisition_Status_Input AT %B4926 : cognex_dataman_380_Acquisition_Status_Input_Layout;

	        // Module cognex_dataman_380/ResultData_128
	        cognex_dataman_380_ResultData_128_Input AT %B4789 : cognex_dataman_380_ResultData_128_Input_Layout;

	        // Module cognex_dataman_380/Results_Status
	        cognex_dataman_380_Results_Status_Input AT %B4925 : cognex_dataman_380_Results_Status_Input_Layout;

	        // Module cognex_dataman_380/Soft_Event_Control
	        cognex_dataman_380_Soft_Event_Control_Input AT %B4929 : cognex_dataman_380_Soft_Event_Control_Input_Layout;

	        // Module cognex_insight_2800/Slot_11_ResultData_250
	        cognex_insight_2800_Slot_11_ResultData_250_Input AT %B4522 : cognex_insight_2800_Slot_11_ResultData_250_Input_Layout;

	        // Module cognex_insight_2800/Slot_12
	        cognex_insight_2800_Slot_12_Input AT %B4272 : cognex_insight_2800_Slot_12_Input_Layout;

	        // Module cognex_insight_2800/Slot_13
	        cognex_insight_2800_Slot_13_Input AT %B4022 : cognex_insight_2800_Slot_13_Input_Layout;

	        // Module cognex_insight_2800/Slot_14
	        cognex_insight_2800_Slot_14_Input AT %B3772 : cognex_insight_2800_Slot_14_Input_Layout;

	        // Module cognex_insight_2800/Slot_2
	        cognex_insight_2800_Slot_2_Input AT %B4776 : cognex_insight_2800_Slot_2_Input_Layout;

	        // Module cognex_insight_2800/Slot_4
	        cognex_insight_2800_Slot_4_Input AT %B4780 : cognex_insight_2800_Slot_4_Input_Layout;

	        // Module cognex_insight_2800/Slot_5
	        cognex_insight_2800_Slot_5_Input AT %B4784 : cognex_insight_2800_Slot_5_Input_Layout;

	        // Module cognex_insight_2800/Slot_6
	        cognex_insight_2800_Slot_6_Input AT %B4788 : cognex_insight_2800_Slot_6_Input_Layout;

	        // Module cognex_insight_7600/Acquisition_Status
	        cognex_insight_7600_Acquisition_Status_Input AT %B5207 : cognex_insight_7600_Acquisition_Status_Input_Layout;

	        // Module cognex_insight_7600/Command_Control
	        cognex_insight_7600_Command_Control_Input AT %B5210 : cognex_insight_7600_Command_Control_Input_Layout;

	        // Module cognex_insight_7600/Inspection_Status
	        cognex_insight_7600_Inspection_Status_Input AT %B5203 : cognex_insight_7600_Inspection_Status_Input_Layout;

	        // Module cognex_insight_7600/ResultData_128
	        cognex_insight_7600_ResultData_128_Input AT %B5071 : cognex_insight_7600_ResultData_128_Input_Layout;

	        // Module cognex_insight_7600/SoftEvent_Control
	        cognex_insight_7600_SoftEvent_Control_Input AT %B5212 : cognex_insight_7600_SoftEvent_Control_Input_Layout;

	        // Module desoutter_cvic_ii/Input_1_byte_1
	        desoutter_cvic_ii_Input_1_byte_1_Input AT %B671 : desoutter_cvic_ii_Input_1_byte_1_Input_Layout;

	        // Module desoutter_cvic_ii/Input_1_byte_2
	        desoutter_cvic_ii_Input_1_byte_2_Input AT %B670 : desoutter_cvic_ii_Input_1_byte_2_Input_Layout;

	        // Module desoutter_cvic_ii/Input_1_word_1
	        desoutter_cvic_ii_Input_1_word_1_Input AT %B664 : desoutter_cvic_ii_Input_1_word_1_Input_Layout;

	        // Module desoutter_cvic_ii/Input_1_word_2
	        desoutter_cvic_ii_Input_1_word_2_Input AT %B658 : desoutter_cvic_ii_Input_1_word_2_Input_Layout;

	        // Module desoutter_cvic_ii/Input_2_word_1
	        desoutter_cvic_ii_Input_2_word_1_Input AT %B666 : desoutter_cvic_ii_Input_2_word_1_Input_Layout;

	        // Module desoutter_cvic_ii/Input_2_word_2
	        desoutter_cvic_ii_Input_2_word_2_Input AT %B660 : desoutter_cvic_ii_Input_2_word_2_Input_Layout;

	        // Module dukaneiqauto/iQ_to_PLC_Inputs
	        dukaneiqauto_iQ_to_PLC_Inputs_Input AT %B518 : dukaneiqauto_iQ_to_PLC_Inputs_Input_Layout;

	        // Module et200sp_CM_4xIO_Link_RF200/CM_4xIO-Link_V2_2_144I_128O_1
	        et200sp_CM_4xIO_Link_RF200_CM_4xIO_Link_V2_2_144I_128O_1_Input AT %B162 : et200sp_CM_4xIO_Link_RF200_CM_4xIO_Link_V2_2_144I_128O_1_Input_Layout;

	        // Module et200sp/CpPtp
	        et200sp_CpPtp_Input AT %B310 : et200sp_CpPtp_Input_Layout;

	        // Module festo_cmmtas/DoServo
	        festo_cmmtas_DoServo_SiemensTelegram111_PZD_12_12_Input AT %B5263 : festo_cmmtas_DoServo_SiemensTelegram111_PZD_12_12_Input_Layout;

	        festo_cmmtas_DoServo_SiemensTelegram750_PZD_4_1_Input AT %B5287 : festo_cmmtas_DoServo_SiemensTelegram750_PZD_4_1_Input_Layout;

	        // Module keyence_iv3/CommandStatusBits
	        keyence_iv3_CommandStatusBits_Input AT %B2116 : keyence_iv3_CommandStatusBits_Input_Layout;

	        // Module keyence_iv3/DeviceResultBits_1
	        keyence_iv3_DeviceResultBits_1_Input AT %B2112 : keyence_iv3_DeviceResultBits_1_Input_Layout;

	        // Module keyence_iv3/DeviceResultBits_2
	        keyence_iv3_DeviceResultBits_2_Input AT %B760 : keyence_iv3_DeviceResultBits_2_Input_Layout;

	        // Module keyence_iv3/DeviceStatistics
	        keyence_iv3_DeviceStatistics_Input AT %B2068 : keyence_iv3_DeviceStatistics_Input_Layout;

	        // Module keyence_iv3/DeviceStatusWords
	        keyence_iv3_DeviceStatusWords_Input AT %B2096 : keyence_iv3_DeviceStatusWords_Input_Layout;

	        // Module keyence_iv3/PositionAdjustResult
	        keyence_iv3_PositionAdjustResult_Input AT %B2048 : keyence_iv3_PositionAdjustResult_Input_Layout;

	        // Module keyence_iv3/ToolResult_1
	        keyence_iv3_ToolResult_1_Input AT %B2028 : keyence_iv3_ToolResult_1_Input_Layout;

	        // Module keyence_iv3/ToolResult_10
	        keyence_iv3_ToolResult_10_Input AT %B1848 : keyence_iv3_ToolResult_10_Input_Layout;

	        // Module keyence_iv3/ToolResult_11
	        keyence_iv3_ToolResult_11_Input AT %B1828 : keyence_iv3_ToolResult_11_Input_Layout;

	        // Module keyence_iv3/ToolResult_12
	        keyence_iv3_ToolResult_12_Input AT %B1808 : keyence_iv3_ToolResult_12_Input_Layout;

	        // Module keyence_iv3/ToolResult_13
	        keyence_iv3_ToolResult_13_Input AT %B1788 : keyence_iv3_ToolResult_13_Input_Layout;

	        // Module keyence_iv3/ToolResult_14
	        keyence_iv3_ToolResult_14_Input AT %B1768 : keyence_iv3_ToolResult_14_Input_Layout;

	        // Module keyence_iv3/ToolResult_15
	        keyence_iv3_ToolResult_15_Input AT %B1748 : keyence_iv3_ToolResult_15_Input_Layout;

	        // Module keyence_iv3/ToolResult_16
	        keyence_iv3_ToolResult_16_Input AT %B1728 : keyence_iv3_ToolResult_16_Input_Layout;

	        // Module keyence_iv3/ToolResult_17
	        keyence_iv3_ToolResult_17_Input AT %B1708 : keyence_iv3_ToolResult_17_Input_Layout;

	        // Module keyence_iv3/ToolResult_18
	        keyence_iv3_ToolResult_18_Input AT %B1688 : keyence_iv3_ToolResult_18_Input_Layout;

	        // Module keyence_iv3/ToolResult_19
	        keyence_iv3_ToolResult_19_Input AT %B1668 : keyence_iv3_ToolResult_19_Input_Layout;

	        // Module keyence_iv3/ToolResult_2
	        keyence_iv3_ToolResult_2_Input AT %B2008 : keyence_iv3_ToolResult_2_Input_Layout;

	        // Module keyence_iv3/ToolResult_20
	        keyence_iv3_ToolResult_20_Input AT %B1648 : keyence_iv3_ToolResult_20_Input_Layout;

	        // Module keyence_iv3/ToolResult_21
	        keyence_iv3_ToolResult_21_Input AT %B1628 : keyence_iv3_ToolResult_21_Input_Layout;

	        // Module keyence_iv3/ToolResult_22
	        keyence_iv3_ToolResult_22_Input AT %B1608 : keyence_iv3_ToolResult_22_Input_Layout;

	        // Module keyence_iv3/ToolResult_23
	        keyence_iv3_ToolResult_23_Input AT %B1588 : keyence_iv3_ToolResult_23_Input_Layout;

	        // Module keyence_iv3/ToolResult_24
	        keyence_iv3_ToolResult_24_Input AT %B1568 : keyence_iv3_ToolResult_24_Input_Layout;

	        // Module keyence_iv3/ToolResult_25
	        keyence_iv3_ToolResult_25_Input AT %B1548 : keyence_iv3_ToolResult_25_Input_Layout;

	        // Module keyence_iv3/ToolResult_26
	        keyence_iv3_ToolResult_26_Input AT %B1528 : keyence_iv3_ToolResult_26_Input_Layout;

	        // Module keyence_iv3/ToolResult_27
	        keyence_iv3_ToolResult_27_Input AT %B1508 : keyence_iv3_ToolResult_27_Input_Layout;

	        // Module keyence_iv3/ToolResult_28
	        keyence_iv3_ToolResult_28_Input AT %B1488 : keyence_iv3_ToolResult_28_Input_Layout;

	        // Module keyence_iv3/ToolResult_29
	        keyence_iv3_ToolResult_29_Input AT %B1468 : keyence_iv3_ToolResult_29_Input_Layout;

	        // Module keyence_iv3/ToolResult_3
	        keyence_iv3_ToolResult_3_Input AT %B1988 : keyence_iv3_ToolResult_3_Input_Layout;

	        // Module keyence_iv3/ToolResult_30
	        keyence_iv3_ToolResult_30_Input AT %B1448 : keyence_iv3_ToolResult_30_Input_Layout;

	        // Module keyence_iv3/ToolResult_31
	        keyence_iv3_ToolResult_31_Input AT %B1428 : keyence_iv3_ToolResult_31_Input_Layout;

	        // Module keyence_iv3/ToolResult_32
	        keyence_iv3_ToolResult_32_Input AT %B1408 : keyence_iv3_ToolResult_32_Input_Layout;

	        // Module keyence_iv3/ToolResult_33
	        keyence_iv3_ToolResult_33_Input AT %B1388 : keyence_iv3_ToolResult_33_Input_Layout;

	        // Module keyence_iv3/ToolResult_34
	        keyence_iv3_ToolResult_34_Input AT %B1368 : keyence_iv3_ToolResult_34_Input_Layout;

	        // Module keyence_iv3/ToolResult_35
	        keyence_iv3_ToolResult_35_Input AT %B1348 : keyence_iv3_ToolResult_35_Input_Layout;

	        // Module keyence_iv3/ToolResult_36
	        keyence_iv3_ToolResult_36_Input AT %B1328 : keyence_iv3_ToolResult_36_Input_Layout;

	        // Module keyence_iv3/ToolResult_37
	        keyence_iv3_ToolResult_37_Input AT %B1308 : keyence_iv3_ToolResult_37_Input_Layout;

	        // Module keyence_iv3/ToolResult_38
	        keyence_iv3_ToolResult_38_Input AT %B1288 : keyence_iv3_ToolResult_38_Input_Layout;

	        // Module keyence_iv3/ToolResult_39
	        keyence_iv3_ToolResult_39_Input AT %B1268 : keyence_iv3_ToolResult_39_Input_Layout;

	        // Module keyence_iv3/ToolResult_4
	        keyence_iv3_ToolResult_4_Input AT %B1968 : keyence_iv3_ToolResult_4_Input_Layout;

	        // Module keyence_iv3/ToolResult_40
	        keyence_iv3_ToolResult_40_Input AT %B1248 : keyence_iv3_ToolResult_40_Input_Layout;

	        // Module keyence_iv3/ToolResult_41
	        keyence_iv3_ToolResult_41_Input AT %B1228 : keyence_iv3_ToolResult_41_Input_Layout;

	        // Module keyence_iv3/ToolResult_42
	        keyence_iv3_ToolResult_42_Input AT %B1208 : keyence_iv3_ToolResult_42_Input_Layout;

	        // Module keyence_iv3/ToolResult_43
	        keyence_iv3_ToolResult_43_Input AT %B1188 : keyence_iv3_ToolResult_43_Input_Layout;

	        // Module keyence_iv3/ToolResult_44
	        keyence_iv3_ToolResult_44_Input AT %B1168 : keyence_iv3_ToolResult_44_Input_Layout;

	        // Module keyence_iv3/ToolResult_45
	        keyence_iv3_ToolResult_45_Input AT %B1148 : keyence_iv3_ToolResult_45_Input_Layout;

	        // Module keyence_iv3/ToolResult_46
	        keyence_iv3_ToolResult_46_Input AT %B1128 : keyence_iv3_ToolResult_46_Input_Layout;

	        // Module keyence_iv3/ToolResult_47
	        keyence_iv3_ToolResult_47_Input AT %B1108 : keyence_iv3_ToolResult_47_Input_Layout;

	        // Module keyence_iv3/ToolResult_48
	        keyence_iv3_ToolResult_48_Input AT %B1088 : keyence_iv3_ToolResult_48_Input_Layout;

	        // Module keyence_iv3/ToolResult_49
	        keyence_iv3_ToolResult_49_Input AT %B1068 : keyence_iv3_ToolResult_49_Input_Layout;

	        // Module keyence_iv3/ToolResult_5
	        keyence_iv3_ToolResult_5_Input AT %B1948 : keyence_iv3_ToolResult_5_Input_Layout;

	        // Module keyence_iv3/ToolResult_50
	        keyence_iv3_ToolResult_50_Input AT %B1048 : keyence_iv3_ToolResult_50_Input_Layout;

	        // Module keyence_iv3/ToolResult_51
	        keyence_iv3_ToolResult_51_Input AT %B1028 : keyence_iv3_ToolResult_51_Input_Layout;

	        // Module keyence_iv3/ToolResult_52
	        keyence_iv3_ToolResult_52_Input AT %B1008 : keyence_iv3_ToolResult_52_Input_Layout;

	        // Module keyence_iv3/ToolResult_53
	        keyence_iv3_ToolResult_53_Input AT %B988 : keyence_iv3_ToolResult_53_Input_Layout;

	        // Module keyence_iv3/ToolResult_54
	        keyence_iv3_ToolResult_54_Input AT %B968 : keyence_iv3_ToolResult_54_Input_Layout;

	        // Module keyence_iv3/ToolResult_55
	        keyence_iv3_ToolResult_55_Input AT %B948 : keyence_iv3_ToolResult_55_Input_Layout;

	        // Module keyence_iv3/ToolResult_56
	        keyence_iv3_ToolResult_56_Input AT %B928 : keyence_iv3_ToolResult_56_Input_Layout;

	        // Module keyence_iv3/ToolResult_57
	        keyence_iv3_ToolResult_57_Input AT %B908 : keyence_iv3_ToolResult_57_Input_Layout;

	        // Module keyence_iv3/ToolResult_58
	        keyence_iv3_ToolResult_58_Input AT %B888 : keyence_iv3_ToolResult_58_Input_Layout;

	        // Module keyence_iv3/ToolResult_59
	        keyence_iv3_ToolResult_59_Input AT %B868 : keyence_iv3_ToolResult_59_Input_Layout;

	        // Module keyence_iv3/ToolResult_6
	        keyence_iv3_ToolResult_6_Input AT %B1928 : keyence_iv3_ToolResult_6_Input_Layout;

	        // Module keyence_iv3/ToolResult_60
	        keyence_iv3_ToolResult_60_Input AT %B848 : keyence_iv3_ToolResult_60_Input_Layout;

	        // Module keyence_iv3/ToolResult_61
	        keyence_iv3_ToolResult_61_Input AT %B828 : keyence_iv3_ToolResult_61_Input_Layout;

	        // Module keyence_iv3/ToolResult_62
	        keyence_iv3_ToolResult_62_Input AT %B808 : keyence_iv3_ToolResult_62_Input_Layout;

	        // Module keyence_iv3/ToolResult_63
	        keyence_iv3_ToolResult_63_Input AT %B788 : keyence_iv3_ToolResult_63_Input_Layout;

	        // Module keyence_iv3/ToolResult_64
	        keyence_iv3_ToolResult_64_Input AT %B768 : keyence_iv3_ToolResult_64_Input_Layout;

	        // Module keyence_iv3/ToolResult_7
	        keyence_iv3_ToolResult_7_Input AT %B1908 : keyence_iv3_ToolResult_7_Input_Layout;

	        // Module keyence_iv3/ToolResult_8
	        keyence_iv3_ToolResult_8_Input AT %B1888 : keyence_iv3_ToolResult_8_Input_Layout;

	        // Module keyence_iv3/ToolResult_9
	        keyence_iv3_ToolResult_9_Input AT %B1868 : keyence_iv3_ToolResult_9_Input_Layout;

	        // Module keyence_sr_1000/BusyStatus
	        keyence_sr_1000_BusyStatus_Input AT %B2288 : keyence_sr_1000_BusyStatus_Input_Layout;

	        // Module keyence_sr_1000/CompletionStatus
	        keyence_sr_1000_CompletionStatus_Input AT %B2287 : keyence_sr_1000_CompletionStatus_Input_Layout;

	        // Module keyence_sr_1000/ErrorStatus
	        keyence_sr_1000_ErrorStatus_Input AT %B2286 : keyence_sr_1000_ErrorStatus_Input_Layout;

	        // Module keyence_sr_1000/HandshakeAndGeneralErrorStatus
	        keyence_sr_1000_HandshakeAndGeneralErrorStatus_Input AT %B2289 : keyence_sr_1000_HandshakeAndGeneralErrorStatus_Input_Layout;

	        // Module keyence_sr_1000/MatchingLevelAndTotalEvaluationGradeStatus
	        keyence_sr_1000_MatchingLevelAndTotalEvaluationGradeStatus_Input AT %B2276 : keyence_sr_1000_MatchingLevelAndTotalEvaluationGradeStatus_Input_Layout;

	        // Module keyence_sr_1000/OperationResultStatus
	        keyence_sr_1000_OperationResultStatus_Input AT %B2256 : keyence_sr_1000_OperationResultStatus_Input_Layout;

	        // Module keyence_sr_1000/ResultData_128
	        keyence_sr_1000_ResultData_128_Input AT %B2120 : keyence_sr_1000_ResultData_128_Input_Layout;

	        // Module keyence_sr_1000/TerminalStatus
	        keyence_sr_1000_TerminalStatus_Input AT %B2285 : keyence_sr_1000_TerminalStatus_Input_Layout;

	        // Module keyence_sr_1000/UnstableReadStatus
	        keyence_sr_1000_UnstableReadStatus_Input AT %B2284 : keyence_sr_1000_UnstableReadStatus_Input_Layout;

	        // Module keyence_sr_750/BusyStatus
	        keyence_sr_750_BusyStatus_Input AT %B2458 : keyence_sr_750_BusyStatus_Input_Layout;

	        // Module keyence_sr_750/CompletionStatus
	        keyence_sr_750_CompletionStatus_Input AT %B2457 : keyence_sr_750_CompletionStatus_Input_Layout;

	        // Module keyence_sr_750/ErrorStatus
	        keyence_sr_750_ErrorStatus_Input AT %B2456 : keyence_sr_750_ErrorStatus_Input_Layout;

	        // Module keyence_sr_750/HandshakeAndGeneralErrorStatus
	        keyence_sr_750_HandshakeAndGeneralErrorStatus_Input AT %B2459 : keyence_sr_750_HandshakeAndGeneralErrorStatus_Input_Layout;

	        // Module keyence_sr_750/MatchingLevelAndTotalEvaluationGradeStatus
	        keyence_sr_750_MatchingLevelAndTotalEvaluationGradeStatus_Input AT %B2446 : keyence_sr_750_MatchingLevelAndTotalEvaluationGradeStatus_Input_Layout;

	        // Module keyence_sr_750/OperationResultStatus
	        keyence_sr_750_OperationResultStatus_Input AT %B2426 : keyence_sr_750_OperationResultStatus_Input_Layout;

	        // Module keyence_sr_750/ResultData_128
	        keyence_sr_750_ResultData_128_Input AT %B2290 : keyence_sr_750_ResultData_128_Input_Layout;

	        // Module keyence_sr_750/TerminalStatus
	        keyence_sr_750_TerminalStatus_Input AT %B2455 : keyence_sr_750_TerminalStatus_Input_Layout;

	        // Module keyence_sr_750/UnstableReadStatus
	        keyence_sr_750_UnstableReadStatus_Input AT %B2454 : keyence_sr_750_UnstableReadStatus_Input_Layout;

	        // Module kuka_rb1/DIO512
	        kuka_rb1_DIO512_Input AT %B5897 : kuka_rb1_DIO512_Input_Layout;

	        // Module kuka_rb2/DIO512
	        kuka_rb2_DIO512_Input AT %B5833 : kuka_rb2_DIO512_Input_Layout;

	        // Module mitsubishi_tz535_robot/In_Out_64_byte
	        mitsubishi_tz535_robot_In_Out_64_byte_Input AT %B5769 : mitsubishi_tz535_robot_In_Out_64_byte_Input_Layout;

	        // Module plc_line/A1
	        plc_line_A1_Input AT %B6089 : plc_line_A1_Input_Layout;

	        // Module rexroth_cs351/Input_2_word_1
	        rexroth_cs351_Input_2_word_1_Input AT %B328 : rexroth_cs351_Input_2_word_1_Input_Layout;

	        // Module rexroth_cs351/Input_4_word_1
	        rexroth_cs351_Input_4_word_1_Input AT %B452 : rexroth_cs351_Input_4_word_1_Input_Layout;

	        // Module rexroth_cs351/Input_4_word_10
	        rexroth_cs351_Input_4_word_10_Input AT %B380 : rexroth_cs351_Input_4_word_10_Input_Layout;

	        // Module rexroth_cs351/Input_4_word_11
	        rexroth_cs351_Input_4_word_11_Input AT %B372 : rexroth_cs351_Input_4_word_11_Input_Layout;

	        // Module rexroth_cs351/Input_4_word_12
	        rexroth_cs351_Input_4_word_12_Input AT %B364 : rexroth_cs351_Input_4_word_12_Input_Layout;

	        // Module rexroth_cs351/Input_4_word_13
	        rexroth_cs351_Input_4_word_13_Input AT %B356 : rexroth_cs351_Input_4_word_13_Input_Layout;

	        // Module rexroth_cs351/Input_4_word_14
	        rexroth_cs351_Input_4_word_14_Input AT %B348 : rexroth_cs351_Input_4_word_14_Input_Layout;

	        // Module rexroth_cs351/Input_4_word_15
	        rexroth_cs351_Input_4_word_15_Input AT %B340 : rexroth_cs351_Input_4_word_15_Input_Layout;

	        // Module rexroth_cs351/Input_4_word_16
	        rexroth_cs351_Input_4_word_16_Input AT %B332 : rexroth_cs351_Input_4_word_16_Input_Layout;

	        // Module rexroth_cs351/Input_4_word_2
	        rexroth_cs351_Input_4_word_2_Input AT %B444 : rexroth_cs351_Input_4_word_2_Input_Layout;

	        // Module rexroth_cs351/Input_4_word_3
	        rexroth_cs351_Input_4_word_3_Input AT %B436 : rexroth_cs351_Input_4_word_3_Input_Layout;

	        // Module rexroth_cs351/Input_4_word_4
	        rexroth_cs351_Input_4_word_4_Input AT %B428 : rexroth_cs351_Input_4_word_4_Input_Layout;

	        // Module rexroth_cs351/Input_4_word_5
	        rexroth_cs351_Input_4_word_5_Input AT %B420 : rexroth_cs351_Input_4_word_5_Input_Layout;

	        // Module rexroth_cs351/Input_4_word_6
	        rexroth_cs351_Input_4_word_6_Input AT %B412 : rexroth_cs351_Input_4_word_6_Input_Layout;

	        // Module rexroth_cs351/Input_4_word_7
	        rexroth_cs351_Input_4_word_7_Input AT %B404 : rexroth_cs351_Input_4_word_7_Input_Layout;

	        // Module rexroth_cs351/Input_4_word_8
	        rexroth_cs351_Input_4_word_8_Input AT %B396 : rexroth_cs351_Input_4_word_8_Input_Layout;

	        // Module rexroth_cs351/Input_4_word_9
	        rexroth_cs351_Input_4_word_9_Input AT %B388 : rexroth_cs351_Input_4_word_9_Input_Layout;

	        // Module rexroth_ctrlx_drive/Inputs
	        rexroth_ctrlx_drive_Inputs_P_0_0106_0_0__STO_function__Operating_status_Input AT %B5233 : rexroth_ctrlx_drive_Inputs_P_0_0106_0_0__STO_function__Operating_status_Input_Layout;

	        rexroth_ctrlx_drive_Inputs_S_0_0084_0_0__Torque_force_feedback_value_Input AT %B5231 : rexroth_ctrlx_drive_Inputs_S_0_0084_0_0__Torque_force_feedback_value_Input_Layout;

	        rexroth_ctrlx_drive_Inputs_S_0_0135_0_0__Drive_status_word__Value_Input AT %B5225 : rexroth_ctrlx_drive_Inputs_S_0_0135_0_0__Drive_status_word__Value_Input_Layout;

	        rexroth_ctrlx_drive_Inputs_S_0_0144_0_0__Signal_status_word__Value_Input AT %B5227 : rexroth_ctrlx_drive_Inputs_S_0_0144_0_0__Signal_status_word__Value_Input_Layout;

	        rexroth_ctrlx_drive_Inputs_S_0_0386_0_0__Position_controller__Position_actual_value_Input AT %B5213 : rexroth_ctrlx_drive_Inputs_S_0_0386_0_0__Position_controller__Position_actual_value_Input_Layout;

	        rexroth_ctrlx_drive_Inputs_S_0_0390_0_0__Diagnostic_message__Manufacturer_status_register_Input AT %B5221 : rexroth_ctrlx_drive_Inputs_S_0_0390_0_0__Diagnostic_message__Manufacturer_status_register_Input_Layout;

	        rexroth_ctrlx_drive_Inputs_S_0_0535_0_0__Velocity_controller__Velocity_actual_value_Input AT %B5217 : rexroth_ctrlx_drive_Inputs_S_0_0535_0_0__Velocity_controller__Velocity_actual_value_Input_Layout;

	        rexroth_ctrlx_drive_Inputs_S_0_1720_0_2__Power_supply_control__Status_word_Input AT %B5229 : rexroth_ctrlx_drive_Inputs_S_0_1720_0_2__Power_supply_control__Status_word_Input_Layout;

	        // Module rexroth_indradrive/Input_9_Words
	        rexroth_indradrive_Input_9_Words_Input AT %B5235 : rexroth_indradrive_Input_9_Words_Input_Layout;

	        // Module rexroth_indradrive/ParamCh_5Words
	        rexroth_indradrive_ParamCh_5Words_Input AT %B5253 : rexroth_indradrive_ParamCh_5Words_Input_Layout;

	        // Module rexroth_press/Input_24_Words
	        rexroth_press_Input_24_Words_Input AT %B460 : rexroth_press_Input_24_Words_Input_Layout;

	        // Module rexroth_press/ParamCh_5Words
	        rexroth_press_ParamCh_5Words_Input AT %B508 : rexroth_press_ParamCh_5Words_Input_Layout;

	        // Module rf186c/CM_1
	        rf186c_CM_1_Input AT %B308 : rf186c_CM_1_Input_Layout;

	        // Module rf186c_cyc/CM
	        rf186c_cyc_CM_Input AT %B160 : rf186c_cyc_CM_Input_Layout;

	        // Module rf186c_cyc/RF260R_1
	        rf186c_cyc_RF260R_1_Input AT %B128 : rf186c_cyc_RF260R_1_Input_Layout;

	        // Module rf186c_cyc/RF340R_1
	        rf186c_cyc_RF340R_1_Input AT %B0 : rf186c_cyc_RF340R_1_Input_Layout;

	        // Module rf186c/Reader_1
	        rf186c_Reader_1_Input AT %B306 : rf186c_Reader_1_Input_Layout;

	        // Module ureol2l/1_T2O_State
	        ureol2l_1_T2O_State_Input AT %B5737 : ureol2l_1_T2O_State_Input_Layout;

	        // Module ureol2l/2_T2O_IO
	        ureol2l_2_T2O_IO_Input AT %B5669 : ureol2l_2_T2O_IO_Input_Layout;

	        // Module ureol2l/3_T2O_Joints
	        ureol2l_3_T2O_Joints_Input AT %B5565 : ureol2l_3_T2O_Joints_Input_Layout;

	        // Module ureol2l/4_T2O_TCP
	        ureol2l_4_T2O_TCP_Input AT %B5489 : ureol2l_4_T2O_TCP_Input_Layout;

	        // Module ureol2l/5_T2O_General_Purpose_Bit_Registers
	        ureol2l_5_T2O_General_Purpose_Bit_Registers_Input AT %B5481 : ureol2l_5_T2O_General_Purpose_Bit_Registers_Input_Layout;

	        // Module ureol2l/6_T2O_General_Purpose_Int_Registers
	        ureol2l_6_T2O_General_Purpose_Int_Registers_Input AT %B5385 : ureol2l_6_T2O_General_Purpose_Int_Registers_Input_Layout;

	        // Module ureol2l/7_T2O_General_Purpose_Float_Registers
	        ureol2l_7_T2O_General_Purpose_Float_Registers_Input AT %B5289 : ureol2l_7_T2O_General_Purpose_Float_Registers_Input_Layout;

	        // Module vision_pro/Engine_Control_1
	        vision_pro_Engine_Control_1_Input AT %B3748 : vision_pro_Engine_Control_1_Input_Layout;

	        // Module vision_pro/Engine_Control_2
	        vision_pro_Engine_Control_2_Input AT %B3740 : vision_pro_Engine_Control_2_Input_Layout;

	        // Module vision_pro/Engine_Control_3
	        vision_pro_Engine_Control_3_Input AT %B3732 : vision_pro_Engine_Control_3_Input_Layout;

	        // Module vision_pro/Engine_Control_4
	        vision_pro_Engine_Control_4_Input AT %B3724 : vision_pro_Engine_Control_4_Input_Layout;

	        // Module vision_pro/Result_Data_240_bytes_1
	        vision_pro_Result_Data_240_bytes_1_Input AT %B3484 : vision_pro_Result_Data_240_bytes_1_Input_Layout;

	        // Module vision_pro/Result_Data_240_bytes_2
	        vision_pro_Result_Data_240_bytes_2_Input AT %B3244 : vision_pro_Result_Data_240_bytes_2_Input_Layout;

	        // Module vision_pro/Result_Data_240_bytes_3
	        vision_pro_Result_Data_240_bytes_3_Input AT %B3004 : vision_pro_Result_Data_240_bytes_3_Input_Layout;

	        // Module vision_pro/Result_Data_240_bytes_4
	        vision_pro_Result_Data_240_bytes_4_Input AT %B2764 : vision_pro_Result_Data_240_bytes_4_Input_Layout;

	        // Module vision_pro/Result_Data_240_bytes_5
	        vision_pro_Result_Data_240_bytes_5_Input AT %B2524 : vision_pro_Result_Data_240_bytes_5_Input_Layout;

	        // Module vision_pro/Result_Data_64_bytes_1
	        vision_pro_Result_Data_64_bytes_1_Input AT %B2460 : vision_pro_Result_Data_64_bytes_1_Input_Layout;

	        // Module vision_pro/System_Control
	        vision_pro_System_Control_Input AT %B3756 : vision_pro_System_Control_Input_Layout;

	        // Module zebra/Data88Bin6Bout
	        zebra_Data88Bin6Bout_Input AT %B672 : zebra_Data88Bin6Bout_Input_Layout;

        END_STRUCT;
    END_TYPE
END_NAMESPACE
